{attribute 'qualified_only'}
{attribute 'strict'}
TYPE Surface :
(
	TOP := 1,
	LEFT,
	RIGHT,
	BOTTOM,
	TOP_LEFT,
	TOP_RIGHT,
	BOTTOM_LEFT,
	BOTTOM_RIGHT,
	
	size
)BYTE;
END_TYPE

(* stored: Version 1.1.0.1, ProductVersion 3.1.4024.11
   DUT Surface: Id {6d0ea893-f968-4c3b-b9db-3776692e01d9} *)
